FUNCTION_BLOCK FB_Sequence_Recorder_Test EXTENDS TcUnit.FB_TestSuite

AddOnePosition();
AddTwoPositions();
ClearPositions();
AddTwoClearAddOne();
TryAddDuplicatePosition();
NumberOfPositionsStored();
ZeroPositionsStored();

METHOD AddOnePosition
VAR
	inputBaseAngle : INT := 123;
	inputShoulderAngle : INT := 123;
	inputElbowAngle : INT := 123;
	expectedBaseAngle : INT := 123;
	actualBaseAngle : INT;
	FB_Seq_Rec: FB_Sequence_Recorder;
	recordPosition : BOOL := TRUE;
END_VAR
TEST('TEST: Add one position');

FB_Seq_Rec(
	inputBase:= inputBaseAngle, 
	inputShoulder:= inputShoulderAngle, 
	inputElbow:= inputElbowAngle, 
	recordPosition:= recordPosition, 
	returnPositionAtIndex:= 0, 
	deletePositions:= FALSE, 
	outputBase=> actualBaseAngle, 
	outputShoulder=> , 
	outputElbow=> , 
	numberRecordedPositions=> , 
	ERROR_arrayFull=> );

IF recordPosition THEN
	recordPosition := FALSE;
END_IF

AssertEquals(Expected := expectedBaseAngle,
	Actual := actualBaseAngle,
	Message := 'Position 1 was not recorded');
	
TEST_FINISHED();
END_METHOD

METHOD AddTwoClearAddOne
VAR
	inputBaseAngle1 : INT := 123;
	inputShoulderAngle1 : INT := 123;
	inputElbowAngle1 : INT := 123;
	expectedBaseAngle1 : INT := 123;
	inputBaseAngle2 : INT := 234;
	inputShoulderAngle2 : INT := 234;
	inputElbowAngle2 : INT := 234;
	expectedShoulderAngle2 : INT := 234;
	actualShoulderAngle1 : INT;
	actualShoulderAngle2 : INT;
	FB_Seq_Rec: FB_Sequence_Recorder;
	recordPosition : BOOL := TRUE;
	delete : BOOL := FALSE;
END_VAR
TEST('TEST: Add two, delete, then add one position');

FB_Seq_Rec(
	inputBase:= inputBaseAngle1, 
	inputShoulder:= inputShoulderAngle1, 
	inputElbow:= inputElbowAngle1, 
	recordPosition:= recordPosition, 
	returnPositionAtIndex:= 0, 
	deletePositions:= delete, 
	outputBase=> actualShoulderAngle1, 
	outputShoulder=> , 
	outputElbow=> , 
	numberRecordedPositions=> , 
	ERROR_arrayFull=> );
	
FB_Seq_Rec(
	inputBase:= inputBaseAngle2, 
	inputShoulder:= inputShoulderAngle2, 
	inputElbow:= inputElbowAngle2, 
	recordPosition:= recordPosition, 
	returnPositionAtIndex:= 1, 
	deletePositions:= delete, 
	outputBase=> , 
	outputShoulder=> actualShoulderAngle2, 
	outputElbow=> , 
	numberRecordedPositions=> , 
	ERROR_arrayFull=> );

delete := TRUE;
recordPosition := FALSE;

FB_Seq_Rec(
	inputBase:= inputBaseAngle2, 
	inputShoulder:= inputShoulderAngle2, 
	inputElbow:= inputElbowAngle2, 
	recordPosition:= recordPosition, 
	returnPositionAtIndex:= 1, 
	deletePositions:= delete, 
	outputBase=> , 
	outputShoulder=> actualShoulderAngle2, 
	outputElbow=> , 
	numberRecordedPositions=> , 
	ERROR_arrayFull=> );

delete := FALSE;
recordPosition := TRUE;


FB_Seq_Rec(
	inputBase:= inputBaseAngle2, 
	inputShoulder:= inputShoulderAngle2, 
	inputElbow:= inputElbowAngle2, 
	recordPosition:= recordPosition, 
	returnPositionAtIndex:= 0, 
	deletePositions:= delete, 
	outputBase=> , 
	outputShoulder=> actualShoulderAngle2, 
	outputElbow=> , 
	numberRecordedPositions=> , 
	ERROR_arrayFull=> );	

AssertEquals(Expected := expectedShoulderAngle2,
	Actual := actualShoulderAngle2,
	Message := 'Wrong value returned');
	
TEST_FINISHED();
END_METHOD

METHOD AddTwoPositions
VAR
	inputBaseAngle1 : INT := 123;
	inputShoulderAngle1 : INT := 123;
	inputElbowAngle1 : INT := 123;
	expectedBaseAngle1 : INT := 123;
	inputBaseAngle2 : INT := 234;
	inputShoulderAngle2 : INT := 234;
	inputElbowAngle2 : INT := 234;
	expectedShoulderAngle2 : INT := 234;
	actualShoulderAngle1 : INT;
	actualShoulderAngle2 : INT;
	FB_Seq_Rec: FB_Sequence_Recorder;
	recordPosition : BOOL := TRUE;
END_VAR
TEST('TEST: Add two positions');

FB_Seq_Rec(
	inputBase:= inputBaseAngle1, 
	inputShoulder:= inputShoulderAngle1, 
	inputElbow:= inputElbowAngle1, 
	recordPosition:= recordPosition, 
	returnPositionAtIndex:= 0, 
	deletePositions:= FALSE, 
	outputBase=> actualShoulderAngle1, 
	outputShoulder=> , 
	outputElbow=> , 
	numberRecordedPositions=> , 
	ERROR_arrayFull=> );
	
FB_Seq_Rec(
	inputBase:= inputBaseAngle2, 
	inputShoulder:= inputShoulderAngle2, 
	inputElbow:= inputElbowAngle2, 
	recordPosition:= recordPosition, 
	returnPositionAtIndex:= 1, 
	deletePositions:= FALSE, 
	outputBase=> , 
	outputShoulder=> actualShoulderAngle2, 
	outputElbow=> , 
	numberRecordedPositions=> , 
	ERROR_arrayFull=> );

IF recordPosition THEN
	recordPosition := FALSE;
END_IF

AssertEquals(Expected := expectedShoulderAngle2,
	Actual := actualShoulderAngle2,
	Message := 'Position 2 was not recorded');
	
TEST_FINISHED();
END_METHOD

METHOD ArrayFull
VAR_INPUT
END_VAR
END_METHOD

METHOD ClearPositions : BOOL
VAR
	inputBaseAngle1 : INT := 123;
	inputShoulderAngle1 : INT := 123;
	inputElbowAngle1 : INT := 123;
	expectedBaseAngle1 : INT := 123;
	inputBaseAngle2 : INT := 234;
	inputShoulderAngle2 : INT := 234;
	inputElbowAngle2 : INT := 234;
	expectedShoulderAngle2 : INT := 0;
	actualShoulderAngle1 : INT;
	actualShoulderAngle2 : INT;
	FB_Seq_Rec: FB_Sequence_Recorder;
	recordPosition : BOOL := TRUE;
	delete : BOOL := FALSE;
END_VAR
TEST('TEST: Clear positions');

FB_Seq_Rec(
	inputBase:= inputBaseAngle1, 
	inputShoulder:= inputShoulderAngle1, 
	inputElbow:= inputElbowAngle1, 
	recordPosition:= recordPosition, 
	returnPositionAtIndex:= 0, 
	deletePositions:= FALSE, 
	outputBase=> actualShoulderAngle1, 
	outputShoulder=> , 
	outputElbow=> , 
	numberRecordedPositions=> , 
	ERROR_arrayFull=> );
	
FB_Seq_Rec(
	inputBase:= inputBaseAngle2, 
	inputShoulder:= inputShoulderAngle2, 
	inputElbow:= inputElbowAngle2, 
	recordPosition:= recordPosition, 
	returnPositionAtIndex:= 1, 
	deletePositions:= delete, 
	outputBase=> , 
	outputShoulder=> actualShoulderAngle2, 
	outputElbow=> , 
	numberRecordedPositions=> , 
	ERROR_arrayFull=> );

IF recordPosition THEN
	recordPosition := FALSE;
END_IF

delete := TRUE;

FB_Seq_Rec(
	inputBase:= inputBaseAngle2, 
	inputShoulder:= inputShoulderAngle2, 
	inputElbow:= inputElbowAngle2, 
	recordPosition:= recordPosition, 
	returnPositionAtIndex:= 1, 
	deletePositions:= delete, 
	outputBase=> , 
	outputShoulder=> actualShoulderAngle2, 
	outputElbow=> , 
	numberRecordedPositions=> , 
	ERROR_arrayFull=> );

AssertEquals(Expected := expectedShoulderAngle2,
	Actual := actualShoulderAngle2,
	Message := 'Positions were not deleted');
	
TEST_FINISHED();
END_METHOD

METHOD ErrorIndexOutOfBounds
VAR_INPUT
END_VAR
// Should not be able to input values larger than 9, as it is only possible to store 10 positions in the array (0-9)
//
END_METHOD

METHOD NumberOfPositionsStored : REFERENCE TO FB_Test
VAR
	FB_Seq_Rec: FB_Sequence_Recorder;
	expectedNumberOfPositionsStored : INT := 5;
	actualNumberOfPositionsStored : INT;
END_VAR
TEST('Return number of positions stored');

FB_Seq_Rec(
	inputBase:= 0, 
	inputShoulder:= 0, 
	inputElbow:= 0, 
	recordPosition:= TRUE, 
	returnPositionAtIndex:= 0, 
	deletePositions:= FALSE, 
	outputBase=> , 
	outputShoulder=> , 
	outputElbow=> , 
	numberRecordedPositions=> , 
	ERROR_arrayFull=> );
	
FB_Seq_Rec(
	inputBase:= 1, 
	inputShoulder:= 0, 
	inputElbow:= 0, 
	recordPosition:= TRUE, 
	returnPositionAtIndex:= 0, 
	deletePositions:= FALSE, 
	outputBase=> , 
	outputShoulder=> , 
	outputElbow=> , 
	numberRecordedPositions=> , 
	ERROR_arrayFull=> );
	
FB_Seq_Rec(
	inputBase:= 0, 
	inputShoulder:= 0, 
	inputElbow:= 0, 
	recordPosition:= TRUE, 
	returnPositionAtIndex:= 0, 
	deletePositions:= FALSE, 
	outputBase=> , 
	outputShoulder=> , 
	outputElbow=> , 
	numberRecordedPositions=> , 
	ERROR_arrayFull=> );

// DELETE
FB_Seq_Rec(
	inputBase:= 1, 
	inputShoulder:= 1, 
	inputElbow:= 1, 
	recordPosition:= FALSE, 
	returnPositionAtIndex:= 0, 
	deletePositions:= TRUE, 
	outputBase=> , 
	outputShoulder=> , 
	outputElbow=> , 
	numberRecordedPositions=> , 
	ERROR_arrayFull=> );
	
FB_Seq_Rec(
	inputBase:= 2, 
	inputShoulder:= 2, 
	inputElbow:= 2, 
	recordPosition:= TRUE, 
	returnPositionAtIndex:= 0, 
	deletePositions:= FALSE, 
	outputBase=> , 
	outputShoulder=> , 
	outputElbow=> , 
	numberRecordedPositions=> , 
	ERROR_arrayFull=> );
	
FB_Seq_Rec(
	inputBase:= 3, 
	inputShoulder:= 3, 
	inputElbow:= 3, 
	recordPosition:= TRUE, 
	returnPositionAtIndex:= 0, 
	deletePositions:= FALSE, 
	outputBase=> , 
	outputShoulder=> , 
	outputElbow=> , 
	numberRecordedPositions=> , 
	ERROR_arrayFull=> );
	
FB_Seq_Rec(
	inputBase:= 4, 
	inputShoulder:= 4, 
	inputElbow:= 4, 
	recordPosition:= TRUE, 
	returnPositionAtIndex:= 0, 
	deletePositions:= FALSE, 
	outputBase=> , 
	outputShoulder=> , 
	outputElbow=> , 
	numberRecordedPositions=> , 
	ERROR_arrayFull=> );
	
FB_Seq_Rec(
	inputBase:= 5, 
	inputShoulder:= 5, 
	inputElbow:= 5, 
	recordPosition:= TRUE, 
	returnPositionAtIndex:= 0, 
	deletePositions:= FALSE, 
	outputBase=> , 
	outputShoulder=> , 
	outputElbow=> , 
	numberRecordedPositions=> , 
	ERROR_arrayFull=> );
	
FB_Seq_Rec(
	inputBase:= 6, 
	inputShoulder:= 6, 
	inputElbow:= 6, 
	recordPosition:= TRUE, 
	returnPositionAtIndex:= 0, 
	deletePositions:= FALSE, 
	outputBase=> , 
	outputShoulder=> , 
	outputElbow=> , 
	numberRecordedPositions=> actualNumberOfPositionsStored, 
	ERROR_arrayFull=> );
	
AssertEquals(Expected := expectedNumberOfPositionsStored,
	Actual := actualNumberOfPositionsStored,
	Message := 'Wrong number of positions stored returned');
	
TEST_FINISHED();
END_METHOD

METHOD TryAddDuplicatePosition
VAR
	inputBaseAngle1 : INT := 123;
	inputShoulderAngle1 : INT := 123;
	inputElbowAngle1 : INT := 123;
	expectedBaseAngle1 : INT := 0;
	inputBaseAngle2 : INT := 0;
	inputShoulderAngle2 : INT := 0;
	inputElbowAngle2 : INT := 0;
	expectedResult : BOOL := FALSE;
	actualBaseAngle1 : INT;
	actualShoulderAngle1 : INT;
	actualElbowAngle1 : INT;
	actualBaseAngle2 : INT;
	actualShoulderAngle2 : INT;
	actualElbowAngle2 : INT;
	FB_Seq_Rec: FB_Sequence_Recorder;
	recordPosition : BOOL := TRUE;
	arePositionsDuplicate: BOOL := FALSE;
END_VAR
TEST('TEST: Try add duplicate positions');

FB_Seq_Rec(
	inputBase:= inputBaseAngle1, 
	inputShoulder:= inputShoulderAngle1, 
	inputElbow:= inputElbowAngle1, 
	recordPosition:= recordPosition, 
	returnPositionAtIndex:= 0, 
	deletePositions:= FALSE, 
	outputBase=> actualBaseAngle1, 
	outputShoulder=> actualShoulderAngle1, 
	outputElbow=> actualElbowAngle1, 
	numberRecordedPositions=> , 
	ERROR_arrayFull=> );
	
FB_Seq_Rec(
	inputBase:= inputBaseAngle2, 
	inputShoulder:= inputShoulderAngle2, 
	inputElbow:= inputElbowAngle2, 
	recordPosition:= recordPosition, 
	returnPositionAtIndex:= 1, 
	deletePositions:= FALSE, 
	outputBase=> actualBaseAngle2, 
	outputShoulder=> actualShoulderAngle2, 
	outputElbow=> actualElbowAngle2, 
	numberRecordedPositions=> , 
	ERROR_arrayFull=> );
	
IF (actualBaseAngle1 = actualBaseAngle2) AND (actualShoulderAngle1 = actualShoulderAngle2) AND (actualElbowAngle1 = actualElbowAngle1) THEN
	arePositionsDuplicate := TRUE;
END_IF

AssertEquals(Expected := expectedResult,
	Actual := arePositionsDuplicate,
	Message := 'Not allowed to add duplicate values!');
	
TEST_FINISHED();
END_METHOD

METHOD ZeroPositionsStored
VAR
	inputBaseAngle : INT := 123;
	inputShoulderAngle : INT := 123;
	inputElbowAngle : INT := 123;
	expectedNumberOfPositionsStored : INT := 0;
	actualNumberOfPositionsStored : INT;
	FB_Seq_Rec: FB_Sequence_Recorder;
	recordPosition : BOOL := FALSE;
END_VAR
TEST('TEST: Zero positions added');

FB_Seq_Rec(
	inputBase:= inputBaseAngle, 
	inputShoulder:= inputShoulderAngle, 
	inputElbow:= inputElbowAngle, 
	recordPosition:= recordPosition, 
	returnPositionAtIndex:= 0, 
	deletePositions:= FALSE, 
	outputBase=> , 
	outputShoulder=> , 
	outputElbow=> , 
	numberRecordedPositions=> actualNumberOfPositionsStored, 
	ERROR_arrayFull=> );


AssertEquals(Expected := expectedNumberOfPositionsStored,
	Actual := actualNumberOfPositionsStored,
	Message := 'There are no positions recorrded');
	
TEST_FINISHED();
END_METHOD

END_FUNCTION_BLOCK

(* stored: Version 1.1.0.1, ProductVersion 3.1.4024.13
   POU FB_Sequence_Recorder_Test: Id {f5c2b13f-1378-4b19-a6ca-f4d7d00d8751}, SpecialFunc None
   Method AddOnePosition: Id {250ab92c-fe4b-4de2-89fa-461cfea3cf83}
   Method AddTwoClearAddOne: Id {02463f65-ed15-4150-a2d4-e1a236ab9179}
   Method AddTwoPositions: Id {66c4d13e-c182-461b-8d96-1bf4269358c5}
   Method ArrayFull: Id {f3928984-d735-43f1-8d6a-1440fcb37427}
   Method ClearPositions: Id {03ab6b4d-1a72-4043-b3ca-81bc8d2c5f10}
   Method ErrorIndexOutOfBounds: Id {d5676aca-9d37-409b-abbd-9c56718a4f10}
   Method NumberOfPositionsStored: Id {d14cd669-2d30-4ef8-9b8f-5a4f63e5eb68}
   Method TryAddDuplicatePosition: Id {ffc03e01-d799-4489-b7b1-8122c4070b44}
   Method ZeroPositionsStored: Id {4c065336-aeb8-472c-a310-efdea5a737d7} *)
